// SIMATIC S7-200 project (STEP 7-Micro/WIN), CPU 221 REL 01.10

ORGANIZATION_BLOCK PRINCIPAL:OB1
TITLE=ASTABLE 3S 1S  /  JEVG
BEGIN
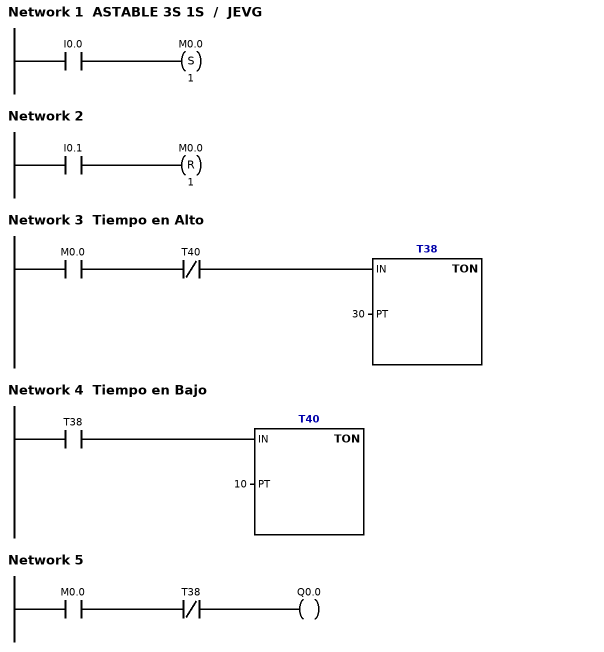
Network 1 // ASTABLE 3S 1S  /  JEVG
LD     I0.0
S      M0.0, 1
Network 2
LD     I0.1
R      M0.0, 1
Network 3 // Tiempo en Alto
LD     M0.0
AN     T40
TON    T38, 30
Network 4 // Tiempo en Bajo
LD     T38
TON    T40, 10
Network 5
LD     M0.0
AN     T38
=      Q0.0
END_ORGANIZATION_BLOCK
